TYPE ST_EquipmentAlarmListDetails :
STRUCT
	FirstAlarm		: POINTER TO ST_EquipmentAlarm;
	AlarmListSize	: DINT; 
END_STRUCT
END_TYPE

(* stored: Version 1.1.0.1
   DUT ST_EquipmentAlarmListDetails: Id {386b1f61-445f-47d6-92a8-768c03d4ce60} *)
